{attribute addProperty BoxType "EL6201-0000-0017"}
{attribute addProperty Id "Slave_17A_DI0BIT10.125129Slave_17A_DI1BIT10.125130Slave_17A_DI2BIT10.125131Slave_17A_DI3BIT10.125132Slave_17B_DI0BIT10.125133Slave_17B_DI1BIT10.125134Slave_17B_DI2BIT10.125135Slave_17B_DI3BIT10.125136"}
{attribute addProperty CRC "4266891903"}
{attribute addProperty SizeInBites "8"}
{attribute addProperty SizeInBytes "1"}
TYPE Slave_17_Inputs_FE539A7F :
STRUCT
	{attribute addProperty Name "Slave_17A_DI0"}
	Slave_17A_DI0 : BIT;
	{attribute addProperty Name "Slave_17A_DI1"}
	Slave_17A_DI1 : BIT;
	{attribute addProperty Name "Slave_17A_DI2"}
	Slave_17A_DI2 : BIT;
	{attribute addProperty Name "Slave_17A_DI3"}
	Slave_17A_DI3 : BIT;
	{attribute addProperty Name "Slave_17B_DI0"}
	Slave_17B_DI0 : BIT;
	{attribute addProperty Name "Slave_17B_DI1"}
	Slave_17B_DI1 : BIT;
	{attribute addProperty Name "Slave_17B_DI2"}
	Slave_17B_DI2 : BIT;
	{attribute addProperty Name "Slave_17B_DI3"}
	Slave_17B_DI3 : BIT;
END_STRUCT
END_TYPE

(* stored: Version 1.2.0.0, ProductVersion 3.1.4024.9
   DUT Slave_17_Inputs_FE539A7F: Id {94315327-1e5e-4400-8d5d-376437eb3dee} *)
